{attribute 'hide_all_locals'}
FUNCTION_BLOCK HaltMover EXTENDS TaskBase
VAR_INPUT
END_VAR
VAR_OUTPUT
END_VAR
VAR
	haltMover : Tc3_McCollisionAvoidance.MC_HaltCA;
	_axis : REFERENCE TO Tc2_MC2.AXIS_REF;
	_HaltMover : BOOL;
END_VAR

CASE State OF
	0:
		IF _HaltMover THEN
			_done := FALSE;
			_error := FALSE;
			_busy := TRUE;
			haltMover.Execute := TRUE;
			IF haltMover.Busy THEN
				State := 10;
				_HaltMover := FALSE;
			END_IF
		END_IF
	
	10:
		IF NOT haltMover.Busy THEN
			IF haltMover.Done THEN
				_done := TRUE;
			ELSIF haltMover.Error THEN
				_error := TRUE;
			END_IF
			_busy := FALSE;
			haltMover.Execute := FALSE;
			State := 0;
		END_IF
END_CASE

haltMover(Axis := _axis);

METHOD Abort : BOOL
haltMover.Execute := FALSE;
_busy := FALSE;
_HaltMover := FALSE;
Abort := TRUE;
State := 0;
END_METHOD

METHOD Execute : BOOL
VAR_INPUT
END_VAR
Execute := _HaltMover := true;
END_METHOD

METHOD FB_init : BOOL
VAR_INPUT
	bInitRetains : BOOL; // if TRUE, the retain variables are initialized (warm start / cold start)
	bInCopyCode : BOOL;  // if TRUE, the instance afterwards gets moved into the copy code (online change)
	axis : reference TO AXIS_REF;
END_VAR
_axis REF= axis;
END_METHOD

END_FUNCTION_BLOCK

(* stored: Version 1.1.0.1, ProductVersion 3.1.4024.12
   POU HaltMover: Id {2df93188-c471-4371-8081-b3d6f1f9ea94}, SpecialFunc None
   Method Abort: Id {227e6d6b-7b18-4f8c-88eb-28da926ffa20}
   Method Execute: Id {1da23db6-3173-436e-9b1a-85386d5bceac}
   Method FB_init: Id {dd4719ba-0246-466b-965a-a67125ef577f} *)
